//---------------------------------------------------------------------------------------------------------------
//
//  HAUD 2024.10.13
//
//
//  fb_StateCollector
//  - base class for process handling
//  - collects states from range of XtsStations
//
//---------------------------------------------------------------------------------------------------------------//
// This SOFTWARE is provided as an Example by THE PROVIDER "as is" and "with all faults." THE PROVIDER makes no  //
// representations or warranties of any kind concerning the safety, suitability, lack of viruses, inaccuracies,  //
// typographical errors, or other harmful components of this SOFTWARE. There are inherent dangers in the use of  //
// any software, and you are solely responsible for determining whether this SOFTWARE is compatible with your    //
// equipment and other software installed on your equipment. You are also solely responsible for the protection  //
// of your equipment and backup of your data, and THE PROVIDER will not be liable for any damages you may suffer //
// in connection with using, modifying, or distributing this SOFTWARE.                                           //
//---------------------------------------------------------------------------------------------------------------//
FUNCTION_BLOCK ABSTRACT fb_StationCollector
VAR
  {info ' extend/add enum members to E_INSTANCE as you need them '}
  _nProcessId     : E_INSTANCE; // whoami

  _eCheck             : E_PROCESS_CHECK;
  _nStationCount      : UINT;

  _nStationFirst,
  _nStationLast       : UINT; // closed range of XtsStations

  // ctrl / state datafields for extern control
  _stStationCtrl      : REFERENCE TO ARRAY[1..MAX_STATION] OF ST_STATION_CTRL;   // control for extern to write
  _stStationState     : REFERENCE TO ARRAY[1..MAX_STATION] OF ST_STATION_STATE;  // state for extern to read

  // mover info datafield
  _MoverInfo          : REFERENCE TO ARRAY[1..MAX_MOVER] OF ST_MOVER_INFO;

  // One Process    - multiple XtsStations
  // One XtsStation - One Mover
  //
  // state words for XtsStations in my range
  {attribute 'displaymode':='bin'}
  _wStateDisable      : T_PROCESS;
  {attribute 'displaymode':='bin'}
  _wStateEnable       : T_PROCESS;
  {attribute 'displaymode':='bin'}
  _wStateEnter        : T_PROCESS;
  {attribute 'displaymode':='bin'}
  _wStateStart        : T_PROCESS;
  {attribute 'displaymode':='bin'}
  _wStateDone         : T_PROCESS;
  {attribute 'displaymode':='bin'}
  _wStateNest         : T_PROCESS;
  {attribute 'displaymode':='bin'}
  _wStateOut          : T_PROCESS;
  {attribute 'displaymode':='bin'}
  _wStateGone         : T_PROCESS;
  {attribute 'displaymode':='bin'}
  _wError             : T_PROCESS;
  {attribute 'displaymode':='bin'}
  _wErrorFatal        : T_PROCESS;

  // One Process    - multiple XtsStations
  // One XtsStation - One Mover
  //

  // important state infos from XtsStations
  _nMoverIdQueue,
  _nStationQueue              : ARRAY[1..SIZEOF(T_PROCESS)*8] OF UINT; // single queues from sub stations
  _nProcessQueue              : UINT; // sum of all sub station queues

  _AllStationMoverPerMinute   : UINT;
  _tonPartsPerMinute          : Tc2_Standard.TON;

  _nMoverCountTotal           : UDINT;

  _stMsg                      : ST_Message;
  _MessageLevel               : E_MessageType;
END_VAR

METHOD PUBLIC BitDel : T_PROCESS
VAR_INPUT
  inVal   : T_PROCESS;
  bitNo   : DINT;
END_VAR
VAR
  wConst : T_PROCESS := 1;
END_VAR
IF ( inVal AND SHL( wConst,TO_SINT(bitNo) MOD TO_INT(SIZEOF(T_PROCESS)*8) ) ) > 0 THEN
  BitDel := inVal XOR (SHL( wConst,TO_SINT(bitNo) MOD TO_INT(SIZEOF(T_PROCESS)*8) ));
ELSE
  BitDel := inVal;
END_IF
END_METHOD

METHOD PUBLIC BitGet : BOOL
VAR_INPUT
  inVal   : T_PROCESS;
  bitNo   : DINT;
END_VAR
VAR
  wConst : T_PROCESS := 1;
END_VAR
IF ( inVal AND SHL( wConst,TO_SINT(bitNo) MOD TO_INT(SIZEOF(T_PROCESS)*8) ) ) > 0
THEN
  BitGet := TRUE;
ELSE
  BitGet := FALSE;
END_IF
END_METHOD

METHOD PUBLIC BitSet : T_PROCESS
VAR_INPUT
  inVal   : T_PROCESS;
  bitNo   : DINT;
END_VAR
VAR
  wConst  : T_PROCESS := 1;
END_VAR
BitSet := inVal OR SHL( wConst,TO_SINT(bitNo) MOD TO_INT(SIZEOF(T_PROCESS)*8) );
END_METHOD

METHOD BitsToString : STRING(SIZEOF(T_PROCESS)*8) // T_PROCESS to string
VAR_INPUT
  inVal       : T_PROCESS;
END_VAR
VAR
  _nx         : DINT;
  _str        : STRING(SIZEOF(T_PROCESS)*8);
END_VAR
FOR _nx := ((SIZEOF(inVal)*8)) TO 1 BY(-1)
DO
  IF (BitGet(inVal, _nx-1))
  THEN
    _str     := concat(_str, '1');
  ELSE
    _str     := concat(_str, '0');
  END_IF
END_FOR

BitsToString := _str;
END_METHOD

METHOD Check : BOOL
VAR_INPUT
END_VAR

IF NOT (_nStationLast > 0)
THEN
  _eCheck             := E_PROCESS_CHECK.STATION_LAST_ZERO;
  RETURN;
END_IF

IF NOT (_nStationFirst > 0)
THEN
  _eCheck             := E_PROCESS_CHECK.STATION_FIRST_ZERO;

  _stMsg.eType        := E_MessageType.eMessageWarning;
  _stMsg.eSubdevice   := e_Subdevice.Process_StationCollector;
  _stMsg.sText        := TO_STRING(_eCheck);
  f_MessageSet(_stMsg);

  _nStationFirst      := _nStationLast;
END_IF

IF NOT (_nStationLast < MAX_STATION+1)
THEN
  _eCheck         := E_PROCESS_CHECK.STATION_LAST_MAX;
  RETURN;
END_IF

IF NOT (_nStationFirst < MAX_STATION+1)
THEN
  _eCheck         := E_PROCESS_CHECK.STATION_FIRST_MAX;
  RETURN;
END_IF

_nStationCount    := _nStationLast - _nStationFirst + 1;
IF NOT (_nStationCount > 0)
THEN
  _eCheck         := E_PROCESS_CHECK.STATION_COUNT_NEGATIVE;
  RETURN;
END_IF

IF (_nStationCount > SIZEOF(T_PROCESS)*8)
THEN
  _eCheck         := E_PROCESS_CHECK.STATION_COUNT_TOO_HIGH;
  RETURN;
END_IF
//-------------------------------------------------------------------------------------------------
// reference checks
//-------------------------------------------------------------------------------------------------
IF NOT __ISVALIDREF(_MoverInfo)
THEN
  _eCheck         := E_PROCESS_CHECK.REFERENCE_MOVER_INFO_INVALID;
  RETURN;
END_IF

_eCheck           := E_PROCESS_CHECK.CHECK_DONE;
Check             := TRUE;
END_METHOD

METHOD GetMoverInStation : ST_MOVER_INFO // mover in station info
VAR_INPUT
  nStation            : UINT;   // index of GVL_XTS.StationState[nStation]
END_VAR
IF NOT Check() THEN RETURN; END_IF

IF NOT (nStation > 0) OR
   NOT (nStation < MAX_STATION+1)
THEN
  RETURN;
ELSE
  IF NOT (_stStationState[nStation].nMoverId > 0)
  THEN
    RETURN;
  ELSE
    GetMoverInStation           := _MoverInfo[_stStationState[nStation].nMoverId];
  END_IF
END_IF
END_METHOD

METHOD GetStationState : ST_STATION_STATE
VAR_INPUT
  nStation            : UINT;   // index of GVL_XTS.StationState[nStation]
END_VAR
IF NOT Check() THEN RETURN; END_IF

IF NOT (nStation > 0) OR
   NOT (nStation < MAX_STATION+1)
THEN
  RETURN;
ELSE
  GetStationState               := _stStationState[nStation];
END_IF
END_METHOD

PROPERTY MoverInfo : REFERENCE TO ARRAY[1..MAX_MOVER] OF ST_MOVER_INFO
SET
_MoverInfo REF= MoverInfo;
END_SET
END_PROPERTY

PROPERTY QueueMoverIDs : ARRAY[1..SIZEOF(T_PROCESS)*8] OF UINT
GET
QueueMoverIDs := _nMoverIdQueue;
END_GET
END_PROPERTY

PROPERTY QueueProcessCount : UINT // sum of all station queues
GET
QueueProcessCount := _nProcessQueue;
END_GET
END_PROPERTY

PROPERTY QueueStationCount : ARRAY[1..SIZEOF(T_PROCESS)*8] OF UINT
GET
QueueStationCount := _nStationQueue;
END_GET
END_PROPERTY

METHOD PROTECTED States // cyclic call for collecting XtsStation state masks
VAR_INST
  _idx    	: UINT;
  _k                    : UINT;
  _rtrigProcess         : ARRAY[1..MAX_STATION] OF Tc2_Standard.R_TRIG;
  _rtrigProcessEnter    : ARRAY[1..MAX_STATION] OF Tc2_Standard.R_TRIG;
  _rtrigProcessStart    : ARRAY[1..MAX_STATION] OF Tc2_Standard.R_TRIG;

  _nMoverPerMinute,
  _nMoverCount,
  _nMoverCountOld       : ARRAY[1..MAX_STATION]  OF UINT;

  _nMoverCountEnter,
  _nMoverCountEnterOld  : ARRAY[1..MAX_STATION]  OF UINT;

  _nMoverCountStart,
  _nMoverCountStartOld  : ARRAY[1..MAX_STATION]  OF UINT;


  _interAllStationsCounter    : UINT;
END_VAR
//-------------------------------------------------------------------------------------------------
//-------------------------------------------------------------------------------------------------
//  HAUD 2024 10 21
//  cyclic call must be implemented by inheriting class 
//  one bit in masks for every XtsStation in process
//
//-------------------------------------------------------------------------------------------------
//-------------------------------------------------------------------------------------------------
_wError                     :=
_wErrorFatal                := 0;

// the sum of movers waiting
_nProcessQueue              := 0;   // calc every plc cycle (see below)

// range checks of _nStationFirst; _nStationLast
IF NOT Check()
THEN
  RETURN;
END_IF

FOR _idx := _nStationLast TO _nStationFirst BY(-1)
DO
  // copy queue for every XtsStation to local for readability (debugging)
  _nStationQueue[(_idx-_nStationFirst+1)] := _stStationState[_idx].nQueue;

  // calc sum of queues for process
  _nProcessQueue                          := _nProcessQueue + _stStationState[_idx].nQueue;

  // get mover ID for all XtsStations in range
  _nMoverIdQueue[(_idx-_nStationFirst+1)] := _stStationState[_idx].nMoverId;

  CASE _stStationCtrl[_idx].Cmd
  OF
    E_STATION_CTRL.STATION_INIT:
      _wStateDisable        := BitDel(_wStateDisable,(_idx - _nStationFirst));
      _wStateEnable         := BitDel(_wStateEnable, (_idx - _nStationFirst));
      _wStateEnter          := BitDel(_wStateEnter,  (_idx - _nStationFirst));
      _wStateStart          := BitDel(_wStateStart,  (_idx - _nStationFirst));
      _wStateDone           := BitDel(_wStateDone,   (_idx - _nStationFirst));
      _wStateNest           := BitDel(_wStateNest,   (_idx - _nStationFirst));
      _wStateOut            := BitDel(_wStateOut,    (_idx - _nStationFirst));
      _wStateGone           := BitDel(_wStateGone,   (_idx - _nStationFirst));
  END_CASE

  CASE _stStationState[_idx].State
  OF
    E_STATION_STATE.STATION_DISABLE:
      _wStateDisable        := BitSet(_wStateDisable,(_idx - _nStationFirst));
      _wStateEnable         := BitDel(_wStateEnable, (_idx - _nStationFirst));
      _wStateOut            := BitDel(_wStateOut,    (_idx - _nStationFirst));
      _wStateGone           := BitDel(_wStateGone,   (_idx - _nStationFirst));
 
    E_STATION_STATE.STATION_ENABLE,
    E_STATION_STATE.STATION_DETECT_MOVER:
      _wStateDisable        := BitDel(_wStateDisable,(_idx - _nStationFirst));
      _wStateEnable         := BitSet(_wStateEnable, (_idx - _nStationFirst));

    E_STATION_STATE.STATION_MOVER_ENTER:
      _wStateEnable         := BitSet(_wStateEnable, (_idx - _nStationFirst));
      _wStateEnter          := BitSet(_wStateEnter,  (_idx - _nStationFirst));

    E_STATION_STATE.STATION_PROCESS_START:
      _wStateStart          := BitSet(_wStateStart,  (_idx - _nStationFirst));
      _wStateNest           := BitDel(_wStateNest,   (_idx - _nStationFirst));

    E_STATION_STATE.STATION_PROCESS_DONE:
      _wStateDone           := BitSet(_wStateDone,   (_idx - _nStationFirst));

    E_STATION_STATE.STATION_CHECK_NEST:
      _wStateStart          := BitDel(_wStateStart,  (_idx - _nStationFirst));
      _wStateDone           := BitDel(_wStateDone,   (_idx - _nStationFirst));
      _wStateNest           := BitSet(_wStateNest,   (_idx - _nStationFirst));

    E_STATION_STATE.STATION_MOVER_OUT:
      _wStateDone           := BitSet(_wStateDone,   (_idx - _nStationFirst));
      _wStateOut            := BitSet(_wStateOut,    (_idx - _nStationFirst));

    E_STATION_STATE.STATION_MOVER_GONE:
      _wStateDisable        := BitDel(_wStateDisable,(_idx - _nStationFirst));
      _wStateEnable         := BitDel(_wStateEnable, (_idx - _nStationFirst));
      _wStateEnter          := BitDel(_wStateEnter,  (_idx - _nStationFirst));
      _wStateStart          := BitDel(_wStateStart,  (_idx - _nStationFirst));
      _wStateDone           := BitDel(_wStateDone,   (_idx - _nStationFirst));
      _wStateNest           := BitDel(_wStateNest,   (_idx - _nStationFirst));
      _wStateOut            := BitDel(_wStateOut,    (_idx - _nStationFirst));

      _wStateGone           := BitSet(_wStateGone, (_idx - _nStationFirst));

    E_STATION_STATE.STATION_ERROR_LIST_STATION_ID_WRONG,  // wrong station ID in mover ticket (nTargetId written by preceeding station/process)
    E_STATION_STATE.STATION_ERROR_OUTFEED_TARGET_INVALID, // write correct target on station Ctrl.nTargetStation
    E_STATION_STATE.STATION_ERROR_INFEED_ERROR,           // clear mover error via Ctrl/State interface and retry on XTS station directly
    E_STATION_STATE.STATION_ERROR_OUTFEED_ERROR:          // clear mover error via Ctrl/State interface and retry on XTS station directly
      _wError               := BitSet(_wError,     (_idx - _nStationFirst));

    E_STATION_STATE.STATION_ERROR_FATAL:
      _wErrorFatal          := BitSet(_wErrorFatal,(_idx - _nStationFirst));

  END_CASE
END_FOR

//-----------------------------------------------------------------------------
// Mover per Minute counter all XtsStations in range
//-----------------------------------------------------------------------------
_nMoverCountTotal           :=
_AllStationMoverPerMinute   := 0; 
//-----------------------------------------------------------------------------
// mover counter
//-----------------------------------------------------------------------------
FOR _k := _nStationLast TO _nStationFirst BY(-1)
DO
  _rtrigProcess[_k](CLK:= ( _stStationCtrl[_k].Cmd = E_STATION_CTRL.STATION_MOVER_OUT));

  IF _rtrigProcess[_k].Q
  THEN
    _nMoverCount[_k]        := _nMoverCount[_k] + 1;

    IF (_MessageLevel > E_MessageType.eMessageVerbose)
    THEN
      _stMsg.eType          := E_MessageType.eMessageSentient;
      _stMsg.eDevice        := e_Device.MetricsXts + TO_UINT(_nProcessId);
                            
      _stMsg.eSubdevice     := e_Subdevice.Process_StationCollector;
      _stMsg.iErrorNumber   := _k;
      _stMsg.sText          := concat('MoverCountStation[ ]: ', TO_STRING(_nMoverCount[_k]));
      _stMsg.sText          := concat(_stMsg.sText, ': E_STATION_CTRL.');
      _stMsg.sText          := concat(_stMsg.sText, TO_STRING(_stStationCtrl[_k].Cmd));
      f_MessageSet(_stMsg);
    END_IF
  END_IF

  _rtrigProcessStart[_k](CLK:= ( _stStationState[_k].State = E_STATION_STATE.STATION_PROCESS_START));

  IF _rtrigProcessStart[_k].Q
  THEN
    _nMoverCountStart[_k]   := _nMoverCountStart[_k] + 1;

    IF (_MessageLevel > E_MessageType.eMessageVerbose)
    THEN
      _stMsg.eType          := E_MessageType.eMessageSentient;
      _stMsg.eDevice        := e_Device.MetricsXts + TO_UINT(_nProcessId);
                            
      _stMsg.eSubdevice     := e_Subdevice.Process_StationCollector;
      _stMsg.iErrorNumber   := _k;
      _stMsg.sText          := concat('MoverCountStation[ ]: ', TO_STRING(_nMoverCountEnter[_k]));
      _stMsg.sText          := concat(_stMsg.sText, ': E_STATION_STATE.');
      _stMsg.sText          := concat(_stMsg.sText, TO_STRING(_stStationState[_k].State));
      f_MessageSet(_stMsg);
    END_IF
  END_IF

  _rtrigProcessEnter[_k](CLK:= ( _stStationCtrl[_k].Cmd = E_STATION_CTRL.STATION_MOVER_ENTER));

  IF _rtrigProcessEnter[_k].Q
  THEN
    _nMoverCountEnter[_k]   := _nMoverCountEnter[_k] + 1;

    IF (_MessageLevel > E_MessageType.eMessageVerbose)
    THEN
      _stMsg.eType          := E_MessageType.eMessageSentient;
      _stMsg.eDevice        := e_Device.MetricsXts + TO_UINT(_nProcessId);
                            
      _stMsg.eSubdevice     := e_Subdevice.Process_StationCollector;
      _stMsg.iErrorNumber   := _k;
      _stMsg.sText          := concat('MoverCountStation[ ]: ', TO_STRING(_nMoverCountEnter[_k]));
      _stMsg.sText          := concat(_stMsg.sText, ': E_STATION_CTRL.');
      _stMsg.sText          := concat(_stMsg.sText, TO_STRING(_stStationCtrl[_k].Cmd));
      f_MessageSet(_stMsg);
    END_IF
  END_IF

  
  IF _tonPartsperMinute.Q
  THEN
    // count every XtsStation in range
    _nMoverPerMinute[_k]    := _nMoverCount[_k] - _nMoverCountOld[_k];
    _nMoverCountOld [_k]    := _nMoverCount[_k];

    _nMoverCountEnterOld [_k]    := _nMoverCountEnter[_k];
    _nMoverCountStartOld [_k]    := _nMoverCountStart[_k];
  END_IF
  // sum up all XtsStations in range
  _AllStationMoverPerMinute := _AllStationMoverPerMinute + _nMoverPerMinute[_k]; 
  _interAllStationsCounter  := _AllStationMoverPerMinute + _nMoverPerMinute[_k];

  // sum up all mover counts in range
  _nMoverCountTotal         := _nMoverCountTotal + _nMoverCount[_k];
END_FOR

IF _tonPartsperMinute.q
THEN
  _tonPartsperMinute(IN:=FALSE);

  IF (_MessageLevel > E_MessageType.eMessageError)
  THEN
    _stMsg.eType            := E_MessageType.eMessageBatch;
    _stMsg.eDevice          := e_Device.MetricsXts + TO_UINT(_nProcessId);
  
    _stMsg.eSubdevice       := e_Subdevice.Process_StationCollector;
    _stMsg.iErrorNumber     := _nMoverCountTotal;
    _stMsg.sText            := concat('MoverCountTotal: ', TO_STRING(_nMoverCountTotal));
    _stMsg.sText            := concat(_stMsg.sText, ': StationLast: ');
    _stMsg.sText            := concat(_stMsg.sText, TO_STRING(_nStationLast));
    _stMsg.sText            := concat(_stMsg.sText, ': StationFirst: ');
    _stMsg.sText            := concat(_stMsg.sText, TO_STRING(_nStationFirst));
    f_MessageSet(_stMsg);
  END_IF
END_IF

_tonPartsperMinute(IN:= TRUE, PT:= T#60S);
END_METHOD

PROPERTY StationCount : UINT
GET
_nStationCount    := _nStationLast - _nStationFirst + 1;
StationCount      := _nStationCount;
END_GET
END_PROPERTY

PROPERTY StationCtrl : reference to ARRAY[1..MAX_STATION] OF ST_STATION_CTRL
SET
_stStationCtrl ref= StationCtrl;
END_SET
END_PROPERTY

PROPERTY StationFirst : uint
GET
StationFirst := _nStationFirst;
END_GET
SET
_nStationFirst := StationFirst;
END_SET
END_PROPERTY

PROPERTY StationLast : uint
GET
StationLast := _nStationLast;
END_GET
SET
_nStationLast := StationLast;
END_SET
END_PROPERTY

PROPERTY StationState : reference to ARRAY[1..MAX_STATION] OF ST_STATION_STATE
SET
_stStationState REF= StationState;
END_SET
END_PROPERTY

METHOD To_T_Process : T_PROCESS // maps (2^nExp)-1 onto T_PROCESS datatype 
VAR_INPUT
  nExp              : BYTE;
END_VAR
VAR
  rVal              : LREAL;
  nTmp              : ULINT; 
  wTmp              : T_PROCESS;
END_VAR
rVal   := TO_LREAL(SEL(nExp > SIZEOF(T_PROCESS)*8, nExp, SIZEOF(T_PROCESS)*8));
nTmp   := TO_ULINT(EXPT(2,rVal)-1);

memcpy(ADR(wtmp), ADR(ntmp), SIZEOF(wtmp));

To_T_Process      := wtmp;
END_METHOD

END_FUNCTION_BLOCK

(* stored: Version 1.1.0.1, ProductVersion 3.1.4026.18
   POU fb_StationCollector: Id {2dc1f5fa-ad5e-46ef-b590-0e1e2dd2e388}, SpecialFunc None
   Folder properties: Id {c5ce3bb8-869f-40b8-a414-c2009ffe56cc}
   Method BitDel: Id {9fa3159e-1717-45de-aa13-e0aeccd74837}
   Method BitGet: Id {fede6eb3-b0d3-49af-85e5-da0659eaf00b}
   Method BitSet: Id {97ed2d75-a3aa-4633-8e6f-0525d8724119}
   Method BitsToString: Id {d040f518-f65d-4793-bdda-9f5b4b05473b}
   Method Check: Id {fb6dc4b9-40cd-408a-8163-7cd4ca2f1726}
   Method GetMoverInStation: Id {cc572b7f-e0d0-424e-b0b0-b379fd0478e3}
   Method GetStationState: Id {b7fc4ff5-2443-428e-b9f7-2a7a1c47ac7a}
   Property MoverInfo: Id {cf62a28d-9468-4ae6-a43b-37fd350a0465}
   Set Set: Id {d1b2c763-e495-40e9-8cb7-cc2d4efae21b}
   Property QueueMoverIDs: Id {cdc56c6b-623d-4fc8-9f8a-69c92b475560}
   Get Get: Id {21a80ed1-022c-44dc-a42d-db583ec8248d}
   Property QueueProcessCount: Id {b4593f38-3f99-4510-b403-e6c016278783}
   Get Get: Id {4313e71c-e077-4e91-bc8f-a4c696463280}
   Property QueueStationCount: Id {2aff4ee2-a827-40fe-ae10-cc7a6329a0ac}
   Get Get: Id {bece7926-60a7-4008-9439-cea17f4fb0e2}
   Method States: Id {a390ee0f-0bc9-4172-9ee2-70281babb672}
   Property StationCount: Id {bbec5067-496d-4247-8253-c81db92c8168}
   Get Get: Id {c1821830-e61d-4b49-aa36-ad10de0c88de}
   Property StationCtrl: Id {6e5d38da-5f20-40ea-8dfc-3d2da85493b2}
   Set Set: Id {95ef5266-c954-46ee-8862-aa770e7a6d13}
   Property StationFirst: Id {7c813fc7-25e1-4034-99b0-cabf3c961465}
   Get Get: Id {6d7dc499-bf2c-45eb-8884-b0cfdccd154d}
   Set Set: Id {f7bc6817-e9ae-44a6-81e5-03bc5d2ff909}
   Property StationLast: Id {105aa0e2-a2f6-4a26-af21-27f3e67d42c5}
   Get Get: Id {a0f2895b-a19f-4fe6-b612-979d73efad0e}
   Set Set: Id {d2b07141-4d6e-4a4f-bde1-cd8d7cd88a12}
   Property StationState: Id {3f366989-a254-460d-8af4-344f08d98e49}
   Set Set: Id {a3909c2b-ce73-4d5c-95c8-e3f1b6cf3764}
   Method To_T_Process: Id {a159cbc2-a5fe-4c16-b032-22ce7f267af9} *)
